PROGRAM MAIN
VAR
	fbSimCell		: FB_SimCell;
END_VAR

fbSimCell();

END_PROGRAM

(* stored: Version 1.1.0.1, ProductVersion 3.1.4024.12
   POU MAIN: Id {978cad62-4036-4e47-9e8a-459f7b1451b8}, SpecialFunc None *)
